FUNCTION F_RoundLREAL : LREAL
VAR_INPUT
	lrValue:					LREAL;
	uiDezimalPlace:	UINT;
END_VAR
VAR
	lrResult:				REAL;
	uiMultiplier:		UINT := 1;
	i:							UINT;
END_VAR

FOR i := 1 TO uiDezimalPlace BY 1 DO
	uiMultiplier := uiMultiplier * 10;
END_FOR

lrResult := TO_REAL(TO_DINT(lrValue * uiMultiplier)) / uiMultiplier;

F_RoundLREAL := lrResult;

END_FUNCTION

(* stored: Version 1.1.0.1, ProductVersion 3.1.4024.12
   POU F_RoundLREAL: Id {3724972c-f60c-4894-9dbb-8536a8db99c3}, SpecialFunc None *)
